FUNCTION F_LeakMonitor_LOCO_1 : FB_LeakMonitor
VAR_INPUT
END_VAR
VAR_OUTPUT
	// Provide stBoundaries output so test functions can reuse the boundaries
	stBoundaries : ST_LeakBoundaries := F_LeakBoundaries();
END_VAR
VAR
	fbLeakMonitor : FB_LeakMonitor;
END_VAR

fbLeakMonitor(
	bLeakDetected := TRUE,
	bCarbideOn := TRUE,
	nLocationResistance := stBoundaries.nLMax2 - 1,
	stBoundaries := stBoundaries,
);

F_LeakMonitor_LOCO_1 := fbLeakMonitor;

END_FUNCTION

(* stored: Version 1.1.0.1, ProductVersion 3.1.4020.14
   POU F_LeakMonitor_LOCO_1: Id {5b6ed2fd-78d0-4541-bbc0-ba1b16217303}, SpecialFunc None *)
